(* PLC project Unnamed, Unknown Unnamed 1 *)
(* stored: creationDateTime 2024-07-25T13:58:10, modificationDateTime 2025-02-06T00:02:25 *)

PROGRAM program0
  VAR
    TANK_1_TEMP AT %IW0 : INT;
    TANK_2_TEMP AT %IW1 : INT;
    TANK_1_LEVEL AT %IW2 : INT;
    TANK_2_LEVEL AT %IW3 : INT;
    FILTER_PUMP_ACTIVE AT %QX0 : BOOL;
    PROGRESSION_PUMP_ACTIVE AT %QX1 : BOOL;
  END_VAR
  VAR CONSTANT
    TANK_FULL : INT := 100;
    PUMP_DELAY : TIME := T#2000ms;
  END_VAR
  VAR
    TOF0 : TOF;
    TOF1 : TOF;
  END_VAR

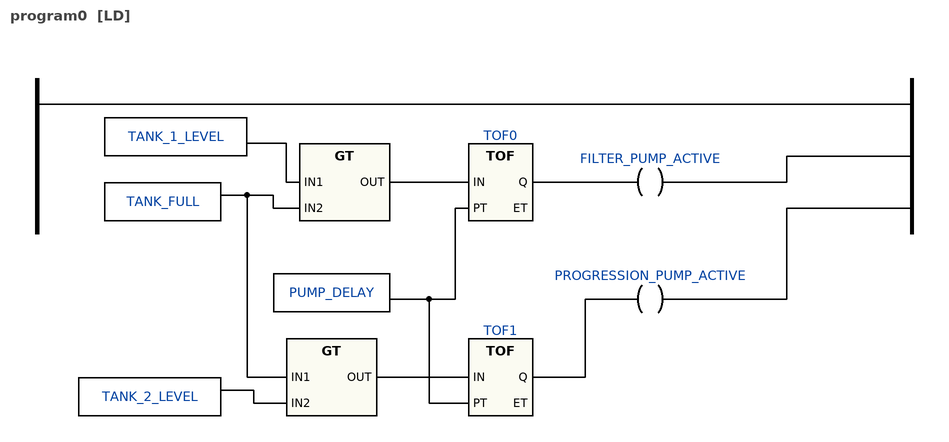
(* LD diagram, written out as Structured Text *)
TOF0(IN := TANK_1_LEVEL > TANK_FULL, PT := PUMP_DELAY);
FILTER_PUMP_ACTIVE := TOF0.Q;
TOF1(IN := TANK_FULL > TANK_2_LEVEL, PT := PUMP_DELAY);
PROGRESSION_PUMP_ACTIVE := TOF1.Q;
END_PROGRAM

CONFIGURATION Config0
  RESOURCE Res0 ON PLC
    TASK task0(INTERVAL := T#20ms, PRIORITY := 0);
    PROGRAM instance0 WITH task0 : program0;
  END_RESOURCE
END_CONFIGURATION
